PROGRAM MAIN
VAR
END_VAR

P_SunriseSunset();
P_WinTime();

P_Doors();
P_Drukknoppen();

P_LightsBerging();
P_LightsBoven();
P_LightsBuiten();
P_LightsHal();
P_LightsKeukenLiving();
P_LightsLeefruimte();

P_Boiler();

P_Temperatures();

P_Screens();

P_Draaipoort();

P_Kwartierpiek();
P_Watermeting();

P_Ventilatie();

P_IoT_Communicator();
P_Sonos();

END_PROGRAM

(* stored: Version 1.1.0.1
   POU MAIN: Id {61422c51-83de-45d6-9242-5ca335c20301}, SpecialFunc None *)
